PROGRAM AssembleParts
VAR
	// Default
	Done: BOOL;
	
	// Scan part id
	AssemblePartId: INT;
	AssemblePartIdReady: BOOL;
	AvailablePartBufferId: INT;
	
	AssembledParts: ARRAY[1..3] OF BOOL;
	
	PartNeedToAssemble: STRING;
	InvalidPart: BOOL;
	Quatity: INT;
	IsUpdateAssemblePartsReady: BOOL;
END_VAR

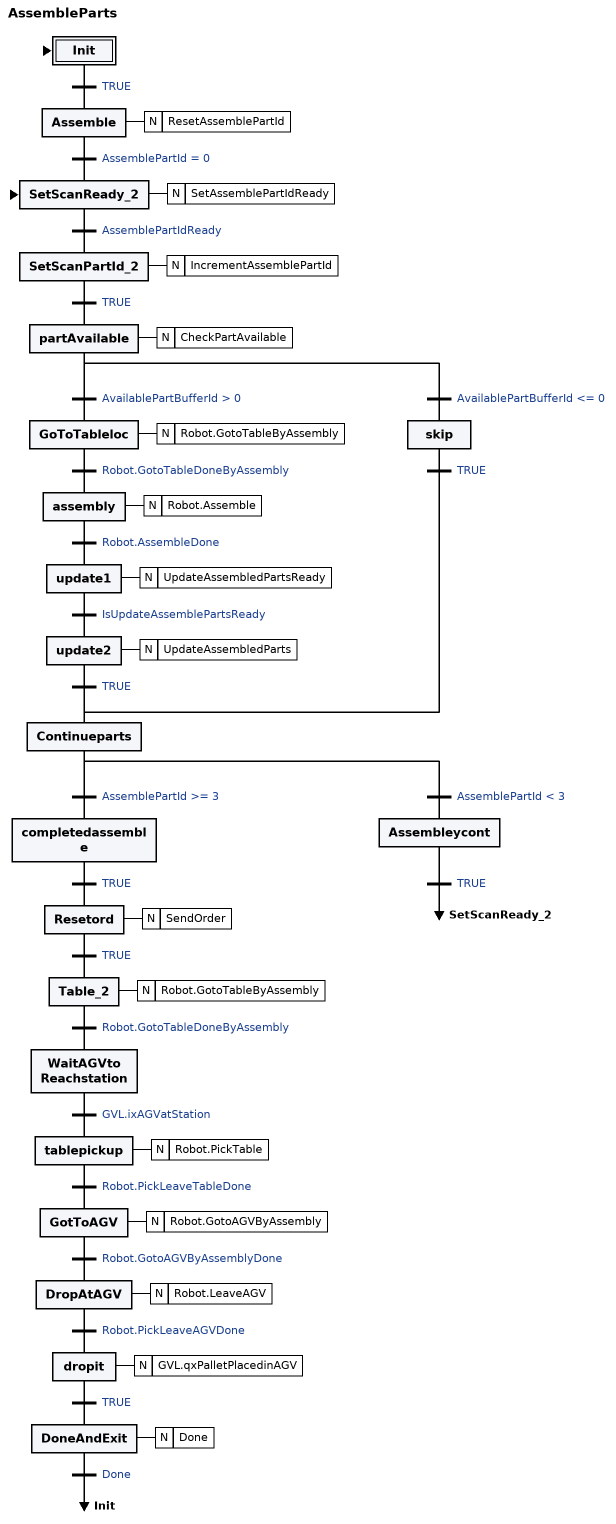
INITIAL_STEP Init:
END_STEP
TRANSITION FROM Init TO Assemble
    := TRUE;
END_TRANSITION
STEP Assemble:
    ResetAssemblePartId(N);
END_STEP
TRANSITION FROM Assemble TO SetScanReady_2
    := AssemblePartId = 0;
END_TRANSITION
STEP SetScanReady_2:
    SetAssemblePartIdReady(N);
END_STEP
TRANSITION FROM SetScanReady_2 TO SetScanPartId_2
    := AssemblePartIdReady;
END_TRANSITION
STEP SetScanPartId_2:
    IncrementAssemblePartId(N);
END_STEP
TRANSITION FROM SetScanPartId_2 TO partAvailable
    := TRUE;
END_TRANSITION
STEP partAvailable:
    CheckPartAvailable(N);
END_STEP
TRANSITION FROM partAvailable TO GoToTableloc
    := AvailablePartBufferId > 0;
END_TRANSITION
STEP GoToTableloc:
    Robot.GotoTableByAssembly(N);
END_STEP
TRANSITION FROM GoToTableloc TO assembly
    := Robot.GotoTableDoneByAssembly;
END_TRANSITION
STEP assembly:
    Robot.Assemble(N);
END_STEP
TRANSITION FROM assembly TO update1
    := Robot.AssembleDone;
END_TRANSITION
STEP update1:
    UpdateAssembledPartsReady(N);
END_STEP
TRANSITION FROM update1 TO update2
    := IsUpdateAssemblePartsReady;
END_TRANSITION
STEP update2:
    UpdateAssembledParts(N);
END_STEP
TRANSITION FROM update2 TO Continueparts
    := TRUE;
END_TRANSITION
TRANSITION FROM partAvailable TO skip
    := AvailablePartBufferId <= 0;
END_TRANSITION
STEP skip:
END_STEP
TRANSITION FROM skip TO Continueparts
    := TRUE;
END_TRANSITION
STEP Continueparts:
END_STEP
TRANSITION FROM Continueparts TO completedassemble
    := AssemblePartId >= 3;
END_TRANSITION
STEP completedassemble:
END_STEP
TRANSITION FROM completedassemble TO Resetord
    := TRUE;
END_TRANSITION
STEP Resetord:
    SendOrder(N);
END_STEP
TRANSITION FROM Resetord TO Table_2
    := TRUE;
END_TRANSITION
STEP Table_2:
    Robot.GotoTableByAssembly(N);
END_STEP
TRANSITION FROM Table_2 TO WaitAGVtoReachstation
    := Robot.GotoTableDoneByAssembly;
END_TRANSITION
STEP WaitAGVtoReachstation:
END_STEP
TRANSITION FROM WaitAGVtoReachstation TO tablepickup
    := GVL.ixAGVatStation;
END_TRANSITION
STEP tablepickup:
    Robot.PickTable(N);
END_STEP
TRANSITION FROM tablepickup TO GotToAGV
    := Robot.PickLeaveTableDone;
END_TRANSITION
STEP GotToAGV:
    Robot.GotoAGVByAssembly(N);
END_STEP
TRANSITION FROM GotToAGV TO DropAtAGV
    := Robot.GotoAGVByAssemblyDone;
END_TRANSITION
STEP DropAtAGV:
    Robot.LeaveAGV(N);
END_STEP
TRANSITION FROM DropAtAGV TO dropit
    := Robot.PickLeaveAGVDone;
END_TRANSITION
STEP dropit:
    GVL.qxPalletPlacedinAGV(N);
END_STEP
TRANSITION FROM dropit TO DoneAndExit
    := TRUE;
END_TRANSITION
TRANSITION FROM Continueparts TO Assembleycont
    := AssemblePartId < 3;
END_TRANSITION
STEP Assembleycont:
END_STEP
TRANSITION FROM Assembleycont TO SetScanReady_2
    := TRUE;
END_TRANSITION
STEP DoneAndExit:
    Done(N);
END_STEP
TRANSITION FROM DoneAndExit TO Init
    := Done;
END_TRANSITION

ACTION CheckPartAvailable:
CASE AssemblePartId OF
	1:
		PartNeedToAssemble := CONCAT (LoadFromAGV.ContainerColor, 'PLATE');
	2:
		IF AssembledParts[1] THEN
			PartNeedToAssemble := CONCAT (LoadFromAGV.ContainerColor, 'CYLINDER');
		ELSE
			PartNeedToAssemble := 'INVALID';
		END_IF
	3:
		IF AssembledParts[1] THEN
			PartNeedToAssemble := CONCAT (LoadFromAGV.ContainerColor, 'OCTAGON');
		ELSE
			PartNeedToAssemble := 'INVALID';
		END_IF
END_CASE
IF GVL.BufferProducts.Storage1.Component = PartNeedToAssemble AND GVL.BufferProducts.Storage1.Quatity > 0 THEN
	AvailablePartBufferId := 1;
ELSIF GVL.BufferProducts.Storage2.Component = PartNeedToAssemble AND GVL.BufferProducts.Storage2.Quatity > 0 THEN
	AvailablePartBufferId := 2;
ELSIF GVL.BufferProducts.Storage3.Component = PartNeedToAssemble AND GVL.BufferProducts.Storage3.Quatity > 0 THEN
	AvailablePartBufferId := 3;
ELSE
	AvailablePartBufferId := -1;
END_IF
END_ACTION

ACTION IncrementAssemblePartId:
IF AssemblePartIdReady THEN
	AssemblePartId := AssemblePartId + 1;
	AssemblePartIdReady := FALSE;
END_IF
END_ACTION

ACTION ResetAssemblePartId:
AssemblePartId := 0;
AssembledParts[1] := FALSE;
AssembledParts[2] := FALSE;
AssembledParts[3] := FALSE;
END_ACTION

ACTION SendOrder:
IF NOT AssembledParts[1] THEN
	GVL.qsOrderFornextAssembly := CONCAT (LoadFromAGV.ContainerColor, 'PLATE');
ELSIF NOT AssembledParts[2] THEN
	GVL.qsOrderFornextAssembly := CONCAT (LoadFromAGV.ContainerColor, 'CYLINDER');
ELSIF NOT AssembledParts[3] THEN
	GVL.qsOrderFornextAssembly := CONCAT (LoadFromAGV.ContainerColor, 'OCTAGON');
ELSE
	GVL.qsOrderFornextAssembly := 'AssembledProduct';
END_IF
END_ACTION

ACTION SetAssemblePartIdReady:
AssemblePartIdReady := TRUE;
END_ACTION

ACTION UpdateAssembledParts:
IF IsUpdateAssemblePartsReady THEN
	CASE AssemblePartId OF
		1:
			AssembledParts[1] := TRUE;
		2:
			AssembledParts[2] := TRUE;
		3:
			AssembledParts[3] := TRUE;
	END_CASE
	CASE AvailablePartBufferId OF
		1:
			GVL.BufferProducts.Storage1.Quatity := GVL.BufferProducts.Storage1.Quatity - 1;
		2:
			GVL.BufferProducts.Storage2.Quatity := GVL.BufferProducts.Storage2.Quatity - 1;
		3:
			GVL.BufferProducts.Storage3.Quatity := GVL.BufferProducts.Storage3.Quatity - 1;
	END_CASE
	IsUpdateAssemblePartsReady := FALSE;
END_IF
END_ACTION

ACTION UpdateAssembledPartsReady:
IsUpdateAssemblePartsReady := TRUE;
END_ACTION

END_PROGRAM

(* stored: Version 1.1.0.1, ProductVersion 3.1.4024.12
   POU AssembleParts: Id {595576f5-0cae-46b2-a7bf-0a6de9a9e03a}, SpecialFunc None
   Action CheckPartAvailable: Id {18441b85-618d-482d-a90e-64c150273747}
   Action IncrementAssemblePartId: Id {c5f758f7-6bf3-474d-adba-73e0ac6e86da}
   Action ResetAssemblePartId: Id {2a9982fa-188e-4ad7-94e2-08f26f9bcc6d}
   Action SendOrder: Id {2afd9be2-421c-412d-9e26-2d7f9c06394a}
   Action SetAssemblePartIdReady: Id {5b8e82b3-15bf-4b2b-81d7-e70954b78143}
   Action UpdateAssembledParts: Id {b048cd18-a54f-4df0-846a-3c0026df27f8}
   Action UpdateAssembledPartsReady: Id {ec795abd-1abc-426c-a80a-a9b91d4f2595} *)
